SUBAPPLICATION logiBUS_AI_Calibrated_Subscribe_VT_OPC (* Remote-Subscribe eines bereits kalibrierten physikalischen Werts (M2M, von der Sensor-Station) -> VT-Anzeige (Q_NumericValue_PHYSA) + lokaler Re-Publish. Die physischen VT-Elemente bleiben hier (dort wo die VT ist): CO/CS-Tasten rufen per CLIENT_0 direkt die ID_CO_METHOD/ID_CS_METHOD auf der Sensor-Station auf (logiBUS_AI_Calibrate_IDA_OPC) - echter Event-zu-Event-Methodenaufruf, kein Toggle/Publish/Subscribe-Umweg (siehe OPC_UA_VERNETZUNG.md Punkt 14). ZERO/SPAN-Referenzwert-Eingabefelder (stObjZero/stObjSpan, siehe v1.8) sind optional - ID_NULL/unbeschrieben lassen, wenn der Sensor feste Referenzwerte hat (Fuellband-Winkel: 0/100 als Literal auf der Sensor-Station), echte Werte durchreichen, wenn der Bediener sie selbst eingibt (Druck: 0/250 bar, kein Kalibrator immer griffbereit). Ersetzt logiBUS_AI_Calibrate_Remote_IDA_OPC: Kalibrierung selbst laeuft jetzt auf der Sensor-Station (logiBUS_AI_Calibrate_IDA_OPC), hier bleibt nur noch Anzeige + VT-Bedienelemente-Weiterleitung. *)
  (* Standard: 61499-2; Description: Copyright (c) 2026 Meisterschulen am Ostbahnhof This program and the accompanying materials are made available under the terms of the Eclipse Public License 2.0 which is available at https://www.eclipse.org/legal/epl-2.0/ SPDX-License-Identifier: EPL-2.0 *)
  (* Version 1.2, 2026-09-17, Franz Höpfinger, Meisterschulen am Ostbahnhof, CO/CS-Weiterleitung von AX_CLIENT_1_0 (Remote-Write) auf AX_PUBLISH_1 (lokaler Publish, Sensor-Station abonniert remote) umgestellt - konsistenter mit der ZERO/SPAN-Weiterleitung (die ohnehin schon so funktioniert, siehe v1.1) und mit dem im Projekt dominanten Subscribe-Richtungsmuster (DRUCK_RAW_M2M etc: der Sensor-seitige Publisher ist immer lokal, die Gegenseite abonniert remote). AX_CLIENT_1_0 war unnoetig - dieser Mechanismus ist im Projekt der Spezialfall fuer 'alleinige Source of Truth'-Kommandos (z.B. Kuehlermotor), nicht das allgemeine Signal-Weiterleitungsmuster. *)
  (* Version 1.3, 2026-09-18, Franz Höpfinger, Meisterschulen am Ostbahnhof, Franz: 'solche Scheiße muss komplett raus' - v1.2s AX_T_FF_SR-Toggle+AX_PUBLISH_1 war selbst wieder ein Event->Pegel->Event-Umweg (Button_IE.IND ist schon ein atomares Event, wird kuenstlich zum Toggle gemacht, nur damit die Sensor-Station es per AX_SUBSCRIBE_1+AX_RF_TRIG wieder zu einem Event zurueckverwandelt). Jetzt: Button_CO/CS.IND direkt auf CLIENT_0.REQ (ACTION=CALL_METHOD), ruft ID_CO_METHOD/ID_CS_METHOD auf der Sensor-Station direkt auf - kein Toggle/Publish/Subscribe/Flankenerkennung mehr noetig. ID_CO_WRITE/ID_CS_WRITE (BOOL-Publish-Adressen) durch ID_CO_CALL/ID_CS_CALL (CALL_METHOD-Adressen) ersetzt. Siehe OPC_UA_VERNETZUNG.md Punkt 14. *)
  (* Version 1.1, 2026-09-17, Franz Höpfinger, Meisterschulen am Ostbahnhof, ZERO/SPAN-Referenzwert-Eingabefelder ergaenzt (uebersehen in v1.0) - ohne diese kann der Kalibrier-Referenzwert (z.B. '0 bar'/'250 bar' bei Druck) nicht mehr von der VT auf STG1 zur jetzt auf der Sensor-Station laufenden CALIBRATE weitergereicht werden. Zwei NumericValue_TO_AR2_OPC-Instanzen (VT-Eingabefeld + OPC-Publish, unveraendert aus dem bisherigen logiBUS_AI_Calibrate_Remote_IDA_OPC-Innenleben wiederverwendet). *)
  (* Version 1.0, 2026-09-17, Franz Höpfinger, Meisterschulen am Ostbahnhof, initial implementation - Franz: 'Analog-Kalibrierung LOKAL, Speichern LOKAL, nur der ENDWERT wird ueber OPC-UA verteilt'. *)
  (* Version 1.5, 2026-09-21, Franz Höpfinger, Meisterschulen am Ostbahnhof, Franz: 'Min Max ist beim Fuellband FEST 0-100 ENDE, das UT braucht keinen Schreibzugriff auf Min/Max' - ZERO/SPAN-Referenzwert-Eingabefelder (stObjZero/stObjSpan/ID_ZERO_READ/WRITE/ID_SPAN_READ/WRITE, SubApps ZeroRef/SpanRef) ersatzlos entfernt. Dieser Typ ist bisher nur fuer Fuellband-Winkel instanziiert, kein anderer Aufrufer betroffen. *)
  (* Version 1.4, 2026-09-21, Franz Höpfinger, Meisterschulen am Ostbahnhof, Neuer Plug CAL_OUT (AR) ergaenzt - durchgereicht von ValueDisplay.VALUE_OUT (AR_M2M_Subscribe_TO_Q_Publish_OPC v1.1) - erster echter Verwendungsfall: Fuellband-Winkel zieht von STG1-Remote-Kalibrierung auf STG2-lokale Kalibrierung um, Befuellautomatik/Fuellband_Oben (beide auf STG1) brauchen den kalibrierten Wert weiterhin als lokalen AR-Plug statt eigenem OPC-UA-Self-Subscribe (Doppel-Self-Subscribe-Vermeidung, wie zuvor ueber AnalogChannel_Fuellband_Winkel.CAL_OUT). *)
  (* Version 1.6, 2026-09-22, Franz Höpfinger, Meisterschulen am Ostbahnhof, Franz: 'Button_IE CLIENT_0 kann eine Subapp werden, das ist ein generelles Muster zum Rufen einer Methode vom VT aus' - Button_CO/Button_CS + CLIENT_CO/CLIENT_CS (Button_IE.IND -> CLIENT_0.REQ) durch je eine Instanz des neuen MyLib::sys::Button_CLIENT_Method_IE ersetzt (TriggerCO/TriggerCS). InputEvent ist dort Parameter statt hartcodiert. *)
  (* Version 1.8, 2026-09-23, Franz Höpfinger, Meisterschulen am Ostbahnhof, ZERO/SPAN-Referenzwert-Eingabefelder wieder ergaenzt (in v1.5 fuer Fuellband entfernt, da dort fest 0/100) - Druck (B20) braucht echte, vom Bediener editierbare Referenzwerte (Franz: 'hier brauchen wir Eingabe, weil man nicht immer einen Kalibrator dabei hat'), kein fester Wert wie bei Fuellband. Neue SubApps ZeroRef/SpanRef (NumericValue_TO_AR2_OPC, identisches Innenleben wie das damals entfernte v1.1/wie im alten logiBUS_AI_Calibrate_Remote_IDA_OPC) - VT-Eingabefeld + optionaler Web-Override hier auf STG1, ID_..._WRITE publiziert den Wert jetzt aber zur Sensor-Station statt ihn nur lokal zu verarbeiten. Optional: stObjZero/stObjSpan default ID_NULL, bestehender Aufrufer (Fuellband) bekommt fuer ID_ZERO/SPAN_READ/WRITE bewusst nie beschriebene Platzhalter-Adressen (wie schon bei FUELLBAND_WINKEL_MINREF_LOC_READ etc.) statt leerem WSTRING-Default, aus Vorsicht vor einer leeren OPC-UA-Adresse zur Laufzeit. *)
  (* Version 1.7, 2026-09-22, Franz Höpfinger, Meisterschulen am Ostbahnhof, Rohwert-Anzeige (RAW/MINRAW/MAXRAW) ergaenzt - fehlte bisher komplett auf STG1: die VT-Objekte existierten schon im Pool und die Sensor-Station (STG2) publiziert sie bereits (siehe logiBUS_AI_Calibrate_2P_IDA_OPC.SUB ID_RAW_WRITE/ID_ZERO_RAW_WRITE/ID_SPAN_RAW_WRITE), aber STG1 hat sie nie abonniert - FUELLBAND_WINKEL_RAW_M2M wurde bei der Umstellung auf lokale Kalibrierung (v1.0-Aera, RemoteSubStrings.gcf v1.19) faelschlich als 'nicht mehr gebraucht' entfernt, MINRAW/MAXRAW-Subscribe gab es nie (kam erst mit der Rohwert-Anzeige-Erweiterung auf der Sensor-Station danach dazu). Drei neue RawDisplay/MinRawDisplay/MaxRawDisplay-Instanzen (AR_M2M_Subscribe_TO_Q_Publish_OPC), analog ValueDisplay fuer CAL - reine Diagnose-Anzeige, kein AR-Plug-Output noetig (VALUE_OUT bleibt unverbunden), aber lokaler Re-Publish (ID_..._WRITE) fuer Web-Mirror/Dashboard-Konsistenz mit CAL. *)
  PACKAGE MyLib::sys;
  IMPORT isobus::UT::Q::const::IDs::ID_NULL;
  IMPORT isobus::UT::io::Button::ButtonActivationCode::BT_PRESSED_LATCHED;
  IMPORT logiBUS::utils::conversion::phys::NumericObjectPool_S;
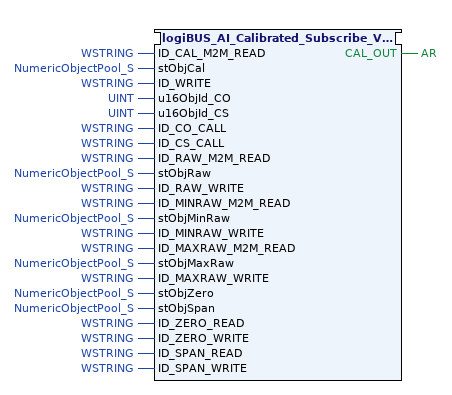
  VAR_INPUT
    ID_CAL_M2M_READ : WSTRING; (* Remote-Subscribe-Adresse des bereits kalibrierten physikalischen Werts (REAL) - Gegenstueck zu ID_CAL_WRITE auf der Sensor-Station (logiBUS_AI_Calibrate_IDA_OPC) *)
    stObjCal : logiBUS::utils::conversion::phys::NumericObjectPool_S := (u16ObjId := ID_NULL, r32Scale := 1.0, i32Offset := 0, u8Decimals := 1); (* Object ID + Scale/Offset/Decimals CNumberVariable (kalibrierter Wert) *)
    ID_WRITE : WSTRING; (* Lokale Re-Publish-Adresse (REAL, ACTION=PUBLISH) fuer weitere lokale Konsumenten auf dieser Station *)
    u16ObjId_CO : UINT := ID_NULL; (* Object ID Taste 'CO' (Kalibrier-Nullpunkt) - physisch hier auf der VT *)
    u16ObjId_CS : UINT := ID_NULL; (* Object ID Taste 'CS' (Kalibrier-Spanne) - physisch hier auf der VT *)
    ID_CO_CALL : WSTRING; (* Remote-Methodenadresse (ACTION=CALL_METHOD) fuer den CO-Trigger - ruft ID_CO_METHOD direkt auf der Sensor-Station auf (logiBUS_AI_Calibrate_IDA_OPC) *)
    ID_CS_CALL : WSTRING; (* Remote-Methodenadresse (ACTION=CALL_METHOD) fuer den CS-Trigger - ruft ID_CS_METHOD direkt auf der Sensor-Station auf (logiBUS_AI_Calibrate_IDA_OPC) *)
    ID_RAW_M2M_READ : WSTRING; (* Remote-Subscribe-Adresse des unkalibrierten Rohwerts (DWORD 0-4095, reine Diagnose-Anzeige) - Gegenstueck zu ID_RAW_WRITE auf der Sensor-Station *)
    stObjRaw : logiBUS::utils::conversion::phys::NumericObjectPool_S := (u16ObjId := ID_NULL, r32Scale := 1.0, i32Offset := 0, u8Decimals := 0); (* Object ID + Scale/Offset/Decimals CNumberVariable (Rohwert-Anzeige) *)
    ID_RAW_WRITE : WSTRING; (* Lokale Re-Publish-Adresse (DWORD, ACTION=PUBLISH) fuer weitere lokale Konsumenten auf dieser Station *)
    ID_MINRAW_M2M_READ : WSTRING; (* Remote-Subscribe-Adresse des Rohwerts am MIN-Kalibrierpunkt (reine Diagnose-Anzeige) - Gegenstueck zu ID_ZERO_RAW_WRITE auf der Sensor-Station *)
    stObjMinRaw : logiBUS::utils::conversion::phys::NumericObjectPool_S := (u16ObjId := ID_NULL, r32Scale := 1.0, i32Offset := 0, u8Decimals := 0); (* Object ID + Scale/Offset/Decimals CNumberVariable (Rohwert-Anzeige am MIN-Kalibrierpunkt) *)
    ID_MINRAW_WRITE : WSTRING; (* Lokale Re-Publish-Adresse (DWORD, ACTION=PUBLISH) fuer weitere lokale Konsumenten auf dieser Station *)
    ID_MAXRAW_M2M_READ : WSTRING; (* Remote-Subscribe-Adresse des Rohwerts am MAX-Kalibrierpunkt (reine Diagnose-Anzeige) - Gegenstueck zu ID_SPAN_RAW_WRITE auf der Sensor-Station *)
    stObjMaxRaw : logiBUS::utils::conversion::phys::NumericObjectPool_S := (u16ObjId := ID_NULL, r32Scale := 1.0, i32Offset := 0, u8Decimals := 0); (* Object ID + Scale/Offset/Decimals CNumberVariable (Rohwert-Anzeige am MAX-Kalibrierpunkt) *)
    ID_MAXRAW_WRITE : WSTRING; (* Lokale Re-Publish-Adresse (DWORD, ACTION=PUBLISH) fuer weitere lokale Konsumenten auf dieser Station *)
    stObjZero : logiBUS::utils::conversion::phys::NumericObjectPool_S := (u16ObjId := ID_NULL, r32Scale := 1.0, i32Offset := 0, u8Decimals := 1); (* Object ID + Scale/Offset/Decimals CNumberVariable (ZERO-Referenzwert, VT-Eingabefeld) - ID_NULL lassen, wenn der Sensor feste Referenzwerte hat (z.B. Fuellband-Winkel) *)
    stObjSpan : logiBUS::utils::conversion::phys::NumericObjectPool_S := (u16ObjId := ID_NULL, r32Scale := 1.0, i32Offset := 0, u8Decimals := 1); (* Object ID + Scale/Offset/Decimals CNumberVariable (SPAN-Referenzwert, VT-Eingabefeld) - ID_NULL lassen, wenn der Sensor feste Referenzwerte hat *)
    ID_ZERO_READ : WSTRING; (* Remote-Subscribe-Adresse ZERO-Referenzwert (REAL, ACTION=SUBSCRIBE) - optionaler Web-Override des VT-Eingabefelds, letzter Schreiber gewinnt *)
    ID_ZERO_WRITE : WSTRING; (* Publish-Adresse ZERO-Referenzwert (REAL, ACTION=PUBLISH) - wird von der Sensor-Station remote abonniert (Gegenstueck zu deren ID_ZERO_READ) *)
    ID_SPAN_READ : WSTRING; (* Remote-Subscribe-Adresse SPAN-Referenzwert (REAL, ACTION=SUBSCRIBE) - optionaler Web-Override des VT-Eingabefelds, letzter Schreiber gewinnt *)
    ID_SPAN_WRITE : WSTRING; (* Publish-Adresse SPAN-Referenzwert (REAL, ACTION=PUBLISH) - wird von der Sensor-Station remote abonniert (Gegenstueck zu deren ID_SPAN_READ) *)
  END_VAR
  PLUGS
    CAL_OUT : adapter::types::unidirectional::AR; (* Nur-Lese-Spiegel des kalibrierten Werts (= ValueDisplay.VALUE_OUT) fuer weitere lokale Konsumenten auf dieser Station, statt eigenem OPC-UA-Self-Subscribe *)
  END_PLUGS
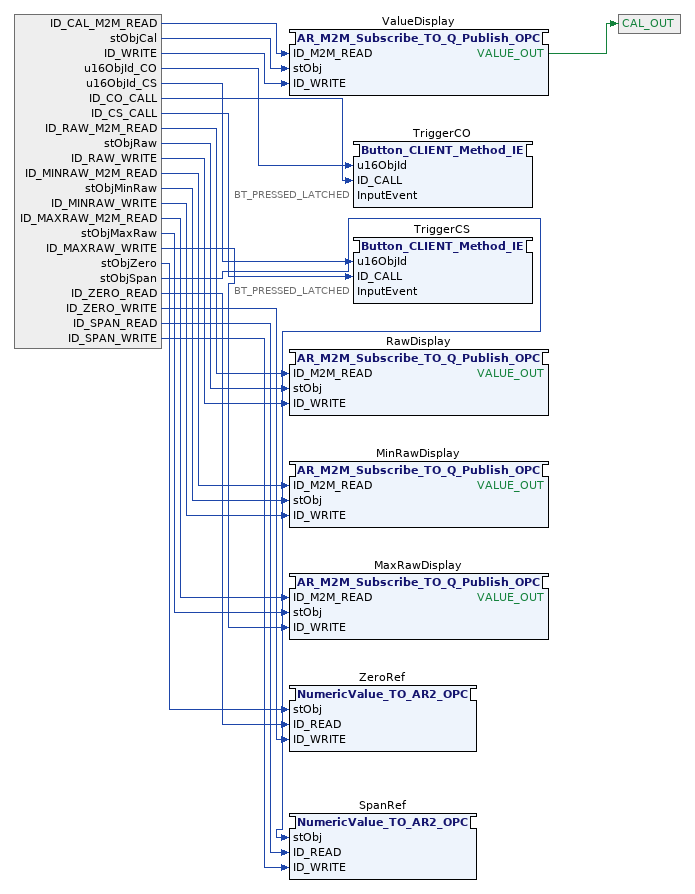
  SUBAPPS
    ValueDisplay : MyLib::sys::AR_M2M_Subscribe_TO_Q_Publish_OPC;
    TriggerCO : MyLib::sys::Button_CLIENT_Method_IE(InputEvent := BT_PRESSED_LATCHED);
    TriggerCS : MyLib::sys::Button_CLIENT_Method_IE(InputEvent := BT_PRESSED_LATCHED);
    RawDisplay : MyLib::sys::AR_M2M_Subscribe_TO_Q_Publish_OPC;
    MinRawDisplay : MyLib::sys::AR_M2M_Subscribe_TO_Q_Publish_OPC;
    MaxRawDisplay : MyLib::sys::AR_M2M_Subscribe_TO_Q_Publish_OPC;
    ZeroRef : MyLib::sys::NumericValue_TO_AR2_OPC;
    SpanRef : MyLib::sys::NumericValue_TO_AR2_OPC;
  END_SUBAPPS
  DATA_CONNECTIONS
    ID_CAL_M2M_READ TO ValueDisplay.ID_M2M_READ;
    stObjCal TO ValueDisplay.stObj;
    ID_WRITE TO ValueDisplay.ID_WRITE;
    u16ObjId_CO TO TriggerCO.u16ObjId;
    u16ObjId_CS TO TriggerCS.u16ObjId;
    ID_CO_CALL TO TriggerCO.ID_CALL;
    ID_CS_CALL TO TriggerCS.ID_CALL;
    ID_RAW_M2M_READ TO RawDisplay.ID_M2M_READ;
    stObjRaw TO RawDisplay.stObj;
    ID_RAW_WRITE TO RawDisplay.ID_WRITE;
    ID_MINRAW_M2M_READ TO MinRawDisplay.ID_M2M_READ;
    stObjMinRaw TO MinRawDisplay.stObj;
    ID_MINRAW_WRITE TO MinRawDisplay.ID_WRITE;
    ID_MAXRAW_M2M_READ TO MaxRawDisplay.ID_M2M_READ;
    stObjMaxRaw TO MaxRawDisplay.stObj;
    ID_MAXRAW_WRITE TO MaxRawDisplay.ID_WRITE;
    stObjZero TO ZeroRef.stObj;
    ID_ZERO_READ TO ZeroRef.ID_READ;
    ID_ZERO_WRITE TO ZeroRef.ID_WRITE;
    stObjSpan TO SpanRef.stObj;
    ID_SPAN_READ TO SpanRef.ID_READ;
    ID_SPAN_WRITE TO SpanRef.ID_WRITE;
  END_CONNECTIONS
  ADAPTER_CONNECTIONS
    ValueDisplay.VALUE_OUT TO CAL_OUT;
  END_CONNECTIONS
END_SUBAPPLICATION
